TYPE EL3152_CHANNEL :
	STRUCT
		
	
	Status 	AT %I* : EL3152_DEV_STATUS;
	Value 	AT %I* : INT;
	
	
	END_STRUCT
END_TYPE

(* stored: Version 1.1.0.1, ProductVersion 3.1.4024.15
   DUT EL3152_CHANNEL: Id {98a8e324-d9ce-4469-97ac-787e9bfa1521} *)
